Universal Robots PolyScope program: implirobot_final.urp

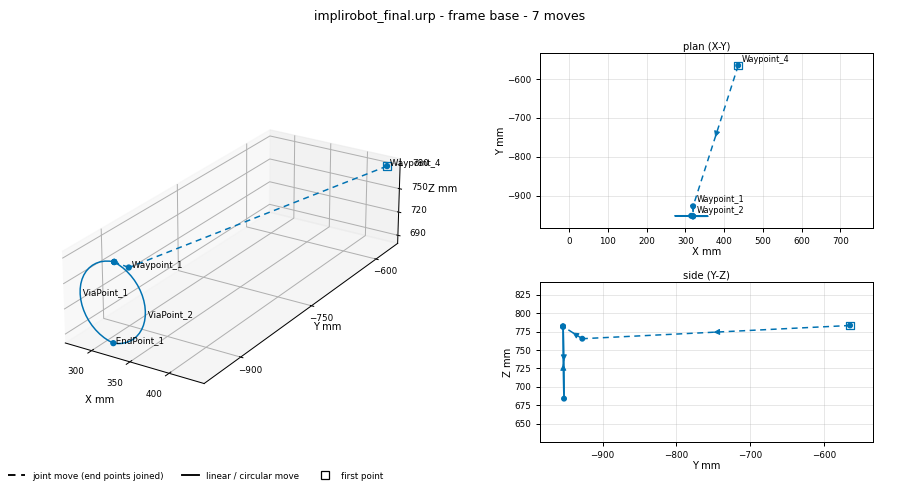
[picture p0: tool path of implirobot_final.urp in frame base, 7 of 9 moves have a stored position in this frame; points joined in program order, loops and branches not executed]
Program implirobot_final (installation=default directory=/programs/usbdisk_0/new folder createdIn=5.12.4.1101661 lastSavedIn=5.12.4.1101661 robotSerialNumber=20205000194)
Calibrated DH parameters: a=[-0.000072, -0.302179, -0.53618, -0.000002, -0.000085, 0]; d=[0.181029, 536.296696, -453.808941, -82.313641, 0.119922, 0.115618]; alpha=[1.57037, -0.000994, -0.002401, 1.569923, -1.570986, 0]; deltaTheta=[0, -1.055132, 6.984537, 0.353782, -0.000001, 0]
Robot Program (runOnlyOnce=false)
  MoveJ speed 60 deg/s, acceleration 80 deg/s^2 (useActiveTCP=true) feature=Base
    Waypoint Waypoint_4: TCP in base x=436.247 y=-564.731 z=783.279 mm, rx=-0.0305 ry=-2.0972 rz=2.0701 rad; joints [-13.309, -87.73, -105.272, -347.036, 4.608, 352.942] deg; TCP offset x=0 y=0 z=160 mm, rx=0 ry=0 rz=0 rad
  MoveJ speed 60 deg/s, acceleration 80 deg/s^2 (useActiveTCP=true) feature=Base
    Waypoint Waypoint_1: TCP in base x=320.041 y=-927.588 z=765.353 mm, rx=0.0291 ry=-2.1159 rz=2.1692 rad; joints [-48.91, -105.454, -88.038, -344.061, 45.344, 352.908] deg
  MoveJ speed 60 deg/s, acceleration 80 deg/s^2 (useActiveTCP=true) feature=Base
    Waypoint Waypoint_2: TCP in base x=319.809 y=-953.656 z=781.919 mm, rx=0.0569 ry=-2.1331 rz=2.1681 rad; joints [-50.579, -106.821, -84.293, -347.284, 48.181, 353.26] deg
    Wait Sleep waitTime=0.3
    MoveP speed 250 mm/s, acceleration 1200 mm/s^2 (blendRadius=0.025 useActiveTCP=true) feature=Base
      Waypoint Waypoint_3: TCP in base x=319.798 y=-953.655 z=781.915 mm, rx=0.0568 ry=-2.1332 rz=2.1681 rad; joints [-50.579, -106.82, -84.294, -347.286, 48.181, 353.262] deg
      CircleMove (OrientationMode=UNCONSTRAINED)
        Waypoint ViaPoint_1: TCP in base x=272.823 y=-952.395 z=730.855 mm, rx=-0.0645 ry=-2.0733 rz=2.1823 rad; joints [-52.196, -107.839, -89.224, -338.323, 45.422, 353.245] deg
        Waypoint EndPoint_1: TCP in base x=314.931 y=-952.311 z=684.111 mm, rx=0.0404 ry=-2.118 rz=2.207 rad; joints [-50.904, -109.524, -91.551, -335.506, 48.859, 353.242] deg
      CircleMove (OrientationMode=UNCONSTRAINED)
        Waypoint ViaPoint_2: TCP in base x=358.018 y=-953.365 z=726.82 mm, rx=0.1146 ry=-2.1452 rz=2.2412 rad; joints [-49.458, -109.303, -87.332, -340.055, 51.168, 353.244] deg
        Waypoint EndPoint_2: TCP in base x=319.821 y=-953.658 z=781.624 mm, rx=0.0571 ry=-2.1333 rz=2.1677 rad; joints [-50.577, -106.822, -84.314, -347.284, 48.176, 353.26] deg
      MoveJ speed 60 deg/s, acceleration 80 deg/s^2 (useActiveTCP=true positionType=JointAngles) feature=Base
        Waypoint Waypoint_5: TCP in base x=319.748 y=-953.653 z=781.896 mm, rx=0.0568 ry=-2.1332 rz=2.1681 rad; joints [-50.581, -106.818, -84.297, -347.285, 48.179, 353.263] deg
